FUNCTION_BLOCK WAVE
  (* Standard: 61499-2 *)
  (* Version 0.1, 2015-00-24, Jin, Jin-PC *)
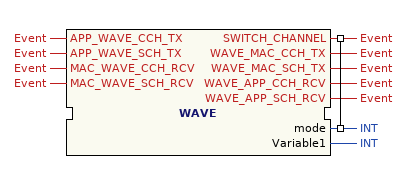
  EVENT_INPUT
    APP_WAVE_CCH_TX;
    APP_WAVE_SCH_TX;
    MAC_WAVE_CCH_RCV;
    MAC_WAVE_SCH_RCV;
  END_EVENT
  EVENT_OUTPUT
    SWITCH_CHANNEL WITH mode;
    WAVE_MAC_CCH_TX;
    WAVE_MAC_SCH_TX;
    WAVE_APP_CCH_RCV;
    WAVE_APP_SCH_RCV;
  END_EVENT
  VAR_OUTPUT
    mode : INT;
    Variable1 : INT;
  END_VAR
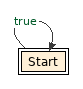
  EC_STATES
    Start;
  END_STATES
  EC_TRANSITIONS
    Start TO Start := true;
  END_TRANSITIONS
END_FUNCTION_BLOCK
